{attribute addProperty BoxType "EJ1914-0000-0017"}
{attribute addProperty Id "Safe_Logic_StateAT %I*USINT811Cycle_CounterAT %I*USINT812"}
{attribute addProperty CRC "2342897971"}
{attribute addProperty SizeInBites "16"}
{attribute addProperty SizeInBytes "2"}
TYPE FSLOGIC_Inputs_8BA5C933 :
STRUCT
	{attribute addProperty Name "Safe_Logic_State"}
	Safe_Logic_State AT %I* : USINT;
	{attribute addProperty Name "Cycle_Counter"}
	Cycle_Counter AT %I* : USINT;
END_STRUCT
END_TYPE

(* stored: Version 1.2.0.0, ProductVersion 3.1.4024.9
   DUT FSLOGIC_Inputs_8BA5C933: Id {892ea40b-d55a-4b45-9ec1-9836a461e4ff} *)
